(*********************************** G.D S.p.A. - Technical Department ***********************************
============= PROGRAM INFO ============
FOLDER:             TBD
MACHINES INVOLVED:  TBD 

============= DESCRIPTION =============
csp machine declaration

============= REVISIONS ===============
Date		Version	 	Author      	Description             
----------	-------		------------  	--------------------------------------------
2019/04/05 	0000.00	 	M.Grasso		Creation of the PRG

**********************************************************************************************************)
(*$R process_ref := prc; $*)
PROGRAM csp_case_tr_accU_ls
VAR
	
	prc:											process;
	prc_path:										STRING;
	
END_VAR

_read_var_input();

_object_manager();

IF NOT objects_running()
THEN
	RETURN;	
END_IF

_read_process_image();

_mode_manager();

_set_runtime_properties();

(********************************* BODY *********************************)
(************************************************************************)

_handle_messages();

_write_output();

ACTION _handle_messages:
;
END_ACTION

ACTION _handle_process_test:
;
END_ACTION

ACTION _mode_manager:
IF process_mode_req_is_pending(prc)
THEN
    process_apply_mode_req_first_step(prc);
    CASE process_get_mode(prc) OF
        MODE_TO_ABSENT:
			;
        MODE_TO_INACTIVE:
			;
        MODE_TO_TEST:
			;
        MODE_TO_OPERATIONAL:
			;
    END_CASE
    process_apply_mode_req_second_step(prc);
END_IF
END_ACTION

ACTION _object_manager:
IF objects_initialization()
THEN
	sub_process_init(
		object_name					:= 'csp_case_tr_accU_ls.prc', 
		process						:= csp_case_topRail_accU.prc, 
		CONVERSION_this				:= prc);
		
	prc_path 						:= process_get_path(prc);
END_IF

IF objects_running()
THEN
	process_cycle(prc);
END_IF
END_ACTION

ACTION _read_process_image:
;
END_ACTION

ACTION _read_var_input:
;
END_ACTION

ACTION _set_runtime_properties:
;
END_ACTION

ACTION _write_output:
;
END_ACTION

END_PROGRAM

(* stored: Version 1.1.0.1, ProductVersion 3.1.4022.12
   POU csp_case_tr_accU_ls: Id {1863a59b-5cb4-4bde-8de7-9d31e9e858de}, SpecialFunc None
   Action _handle_messages: Id {f97c35f3-a05d-4503-8c56-e84e7e61ed6d}
   Action _handle_process_test: Id {b0d93ea6-7733-4433-93e5-5437154038c9}
   Action _mode_manager: Id {eb5e876c-d2af-42e4-9291-1cc86c56b42a}
   Action _object_manager: Id {7ce7ff74-7147-4447-9c65-4666e5628177}
   Action _read_process_image: Id {d4b9fa17-1fa5-47e9-990d-aae40c402bf7}
   Action _read_var_input: Id {e80d81d2-5d7f-4611-8fad-d18eab2b9fd1}
   Action _set_runtime_properties: Id {fab0be1e-f967-481e-97ee-5ac4389eb26e}
   Action _write_output: Id {3722747a-833d-4278-9038-c41eaca1c648} *)
